TYPE uCCDatagram :

UNION
	CCDataStreamHeader: sCCDataStreamHeader;
	CCData: ARRAY[0..63] OF WORD;
END_UNION

END_TYPE

(* stored: Version 1.1.0.1, ProductVersion 3.1.4022.16
   DUT uCCDatagram: Id {4e17725a-d899-4637-a87c-277815c830d3} *)
